(* CoDeSys 2.3.9.50 project: DCMotor_IDS.pro *)
(* Libraries: STANDARD.LIB 5.6.98 12:03:02 *)

(* Task configuration *)
TASK Standard (PRIORITY := 0, INTERVAL := T#10ms);
	MAIN
END_TASK

(* Global variable list: Global_Variables *)
VAR_GLOBAL
	gr_T		: REAL := 0.01;
END_VAR

(* Global variable list: TwinCAT_Configuration *)
(* Generated automatically by TwinCAT - (read only) *)
VAR_CONFIG
	MAIN.b_butYellow AT %IX8.0 : BOOL;
	MAIN.b_butBlue AT %IX8.1 : BOOL;
	MAIN.b_lampRed AT %QX10.0 : BOOL;
	MAIN.b_lampGreen AT %QX10.1 : BOOL;
	MAIN.i_anDisp AT %QB8 : INT;
	MAIN.b_enableMotor AT %QX2.0 : BOOL;
	MAIN.i_motorVoltage AT %QB4 : INT;
	MAIN.ui_encTicks AT %IB2 : UINT;
	MAIN.b_encOver AT %IX4.2 : BOOL;
	MAIN.b_encUnder AT %IX4.3 : BOOL;
END_VAR

(* POU MAIN, ST *)
PROGRAM MAIN
VAR

	b_butYellow		AT %I*	:BOOL;			(* Yellow button *)
	b_butBlue		AT %I*	:BOOL;			(* Blue button *)
	b_lampRed		AT %Q*	:BOOL;			(* Red lamp *)
	b_lampGreen		AT %Q*	:BOOL;			(* Green lamp *)
	i_anDisp		AT %Q*	:INT;			(* Analog meter *)

	b_enableMotor	AT %Q*	:BOOL := TRUE;	(* Motor on/off *)
	i_motorVoltage	AT %Q*	:INT;			(* Motor voltage -24V..+24V coded as -32768..+32767 *)

	ui_encTicks		AT %I*	:UINT;			(* Encoder ticks *)
	b_encOver		AT %I*	:BOOL;			(* Encoder overflow flag, toggles at every overflow *)
	b_encUnder		AT %I*	:BOOL;			(* Encoder underflow flag, toggles at every underflow *)


	ui_deltaTimeMs	:UINT:=10;				(* Encoder sampling time *)
	ui_ticksPerRev	:UINT:=512;				(* Encoder resolution *)


	ui_encTicksOld	:UINT;
	di_deltaTicks	:DINT;
	b_encOverOld	:BOOL;
	b_encUnderOld	:BOOL;
	di_motSpeed		:DINT;

END_VAR
IF b_butYellow = TRUE THEN			(* Turn on with yellow button *)
	b_lampGreen := TRUE;
	b_lampRed := FALSE;
	i_motorVoltage := 10000;
END_IF

IF b_butBLUE = TRUE THEN			(* Turn off*)
	b_lampRed := TRUE;
	b_lampGreen := FALSE;
	i_motorVoltage := 0;
END_IF

di_deltaTicks := ui_encTicks - ui_encTicksOld;	(* Calculate moved track *)
ui_encTicksOld := ui_encTicks;

IF b_encOver <> b_encOverOld THEN			(* Cover overflow *)
	b_encOverOld := b_encOver;
	di_deltaTicks := di_deltaTicks + 65536;
END_IF

IF b_encUnder <> b_encUnderOld THEN		(* Cover underflow *)
	b_encUnderOld := b_encUnder;
	di_deltaTicks := di_deltaTicks - 65536;
END_IF

di_motSpeed := di_deltaTicks *25 / ui_ticksPerRev; 		(* Calculate speed in revolution per seconds *)

i_anDisp := DINT_TO_INT(300 * di_motSpeed);
END_PROGRAM

(* POU chirpSignal, ST *)
FUNCTION_BLOCK chirpSignal
VAR_INPUT
	r_wmin					: REAL;
	r_wmax					: REAL;
	r_ExperimentLength		: REAL;
	r_T						: REAL;
END_VAR
VAR_OUTPUT
	r_Sig	: REAL;
END_VAR
VAR
	(* WORD = 16bit*)
	r_N	: REAL 	:= 0;
	r_k	: REAL	:= 0;
END_VAR
(* Generates Linear Chirp *)
(* w = wmin + kt *)
r_k := (r_wmax - r_wmin) / r_ExperimentLength;		(* Calculate frequency change *)
r_N := (r_ExperimentLength / r_T) + 1;				(* Calculate number of steps *)

r_Sig := COS((r_wmin + r_k * r_N * r_T) * r_T);		(* Calculate next signal value *)
r_N := r_N + 1;										(* Increase next step *)
END_FUNCTION_BLOCK

(* Visualisation GUI
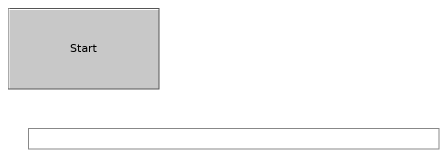
button at (100,160)-(251,241): text "Start"; toggles MAIN.b_testBool
1 more shapes without text or variables
1 elements of other kinds (tables, trends, ...) not read
*)
